TYPE ST_Point :
STRUCT
	x : INT;
	y : INT;
END_STRUCT
END_TYPE

(* stored: Version 1.1.0.1, ProductVersion 3.1.4026.18
   DUT ST_Point: Id {00000000-0000-0000-0000-000000000020} *)
